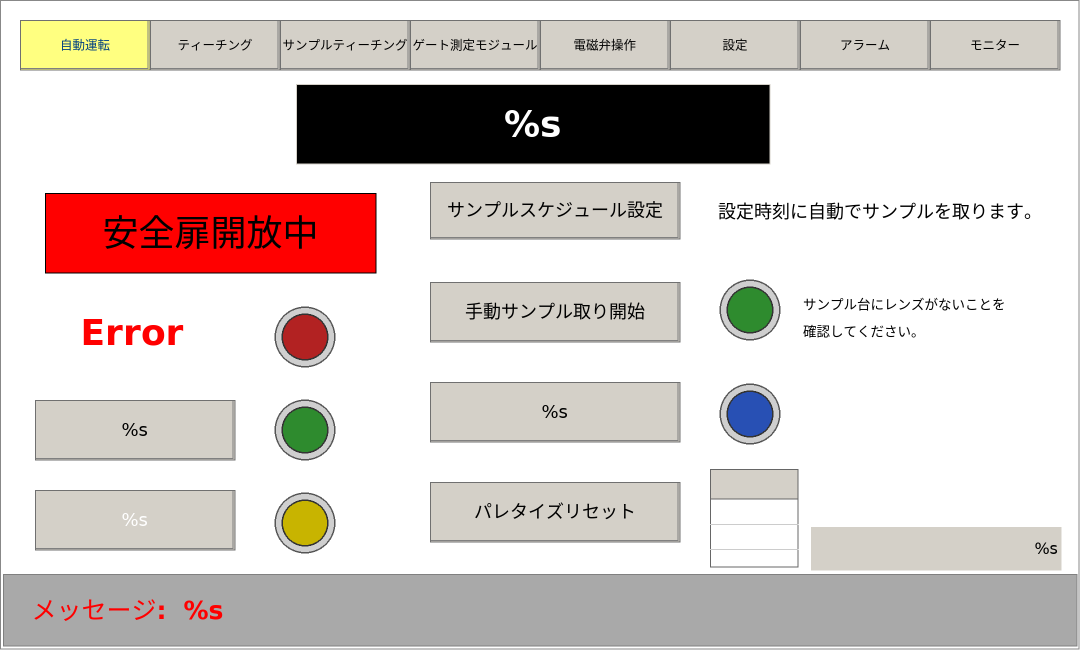
VISUALIZATION s_auto  // 1080x650
    Rectangle (0,0 1080x650)
    Button (35,400 200x60), "%s", text variable: gvl_text.var_auto_runing
        tap gvl_visu.flg_btn_autoModeStart
    Button (35,490 200x60), "%s", text variable: gvl_text.var_stopping, colour toggle: gvl_auto.autoModeStop
        tap gvl_visu.flg_btn_autoModeStop
    Button (430,382 250x60), "%s", text variable: gvl_text.var_trayChangeDone
        toggle gvl_visu.flg_btn_trayChangeDone
    Lamp1 (715,275 70x70), variable: gvl_visu.flg_btn_sample, style: Lamp-Lamp1-Green
    Lamp1 (270,395 70x70), variable: gvl_param.var_currentMode = eP_programMode.auto, style: Lamp-Lamp1-Green
    Lamp1 (270,488 70x70), variable: gvl_param.var_currentMode = eP_programMode.manual, style: Lamp-Lamp1-Yellow
    Lamp1 (270,302 70x70), variable: gvl_param.var_currentMode = eP_programMode.error, invisible if: gvl_param.var_currentMode <> eP_programMode.error, style: Lamp-Lamp1-Red
    Label (42,293 180x79), "Error", invisible if: gvl_param.var_currentMode <> eP_programMode.error
    Lamp1 (715,379 70x70), variable: gvl_visu.flg_btn_trayChangeDone, style: Lamp-Lamp1-Blue
    RoundedRectangle (811,527 250x43), "%s", text variable: gvl_visu.var_DT
    Button (430,282 250x60), "手動サンプル取り開始"
        toggle gvl_visu.flg_btn_sample
    Rectangle (296,84 474x80), "%s", text variable: gvl_param.var_productInfo[gvl_param.var_currentProductID].name
    Rectangle (3,574 1074x72), "メッセージ: %s", text variable: gvl_visu.var_msg
    Button (430,482 250x60), "パレタイズリセット"
        OnMouseClick: OpenDialog Dialog=d_palletizeReset, OpenModal=True, OpenCentered=True
    Table (710,469 88x98), data array: gvl_auto.pocketNo
        p3854506369: gvl_auto.pocketNo[INDEX]
    Button (20,20 130x50), "自動運転"
        OnMouseClick: change screen: s_auto
    Button (150,20 130x50), "ティーチング"
        OnMouseClick: change screen: s_teaching1
    Button (670,20 130x50), "設定"
        OnMouseClick: change screen: s_setting
    Button (540,20 130x50), "電磁弁操作"
        OnMouseClick: change screen: s_manual
    Button (410,20 130x50), "ゲート測定モジュール"
        OnMouseClick: change screen: s_gm_teaching
    Button (800,20 130x50), "アラーム", colour toggle: gvl_io.flg_signalTowerRed
        OnMouseClick: change screen: s_alarm
    Button (280,20 130x50), "サンプルティーチング"
        OnMouseClick: change screen: s_sample
    Button (430,182 250x57), "サンプルスケジュール設定"
        OnMouseClick: OpenDialog Dialog=d_sampleSchedule, OpenModal=True, OpenCentered=True
    Label (715,185 363x54), "設定時刻に自動でサンプルを取ります。"
    Button (930,20 130x50), "モニター"
        OnMouseClick: change screen: s_monitor
    Label (800,280 250x50), "サンプル台にレンズがないことを"
    Rectangle (45,193 331x80), "安全扉開放中", text variable: gvl_io.flg_frontSaftyDoor or gvl_param.var_currentMode <> eP_programMode.auto, invisible if: gvl_io.flg_frontSaftyDoor or gvl_param.var_currentMode <> eP_programMode.auto
    Label (800,307 250x50), "確認してください。"
END_VISUALIZATION

(* stored: Version 1.1.0.1, ProductVersion 3.1.4024.11
   Visu s_auto: Id {4398e26c-8905-4d9c-9981-c42656d5b02a} *)
